// TIA Portal V20 export
// export: Created 2025-12-01T14:56:22.6904925Z, ExportSetting None, DisplayName Totally Integrated Automation Portal, DisplayVersion V20 Update 3, DisplayName TIA Portal Openness, DisplayVersion V20 Update 3, DisplayName TIA Portal Version Control Interface, DisplayVersion V20 Update 3, DisplayName STEP 7 Professional, DisplayVersion V20 Update 3, DisplayName STEP 7 Safety, DisplayVersion V20 Update 2, DisplayName WinCC Basic/Comfort/Advanced, DisplayVersion V20 Update 3, DisplayName WinCC Professional, DisplayVersion V20 Update 3, DisplayName WinCC Unified, DisplayVersion V20 Update 3
TYPE "MoviManualMesa_Eraman"
   STRUCT
      Avance_Rod : Bool;
      Retroceso_Rod : Bool;
      Avance_Cad_TR1 : Bool;
      Retroceso_Cad_TR1 : Bool;
      Subir_TR1 : Bool;
      Bajar_TR1 : Bool;
      Subir_TP1 : Bool;
      Bajar_TP1 : Bool;
      Avance_Cad_TR2 : Bool;
      Retroceso_Cad_TR2 : Bool;   // ...
      Subir_TR2 : Bool;   // ...
      Bajar_TR2 : Bool;   // ...
      Subir_TP2 : Bool;   // ...
      Bajar_TP2 : Bool;   // ...
      Subir_TPS3 : Bool;   // ...
      Bajar_TPS3 : Bool;   // ...
      Subir_TPE1 : Bool;   // ...
      Bajar_TPE1 : Bool;   // ...
      Byte2_bit2 : Bool;   // ...
      Byte2_bit3 : Bool;   // ...
      Byte2_bit4 : Bool;   // ...
      Byte2_bit5 : Bool;   // ...
      Byte2_bit6 : Bool;   // ...
      Byte2_bit7 : Bool;   // ...
      Avance_Cad_Ambos_Transfers : Bool;   // ...
      Retroceso_Cad_Ambos_Transfers : Bool;   // ...
      "Avance+Siguiente_Cad_TR1" : Bool;   // ...
      "Retroceso+Siguiente_Cad_TR1" : Bool;   // ...
      "Avance+Anterior_Cad_TR1" : Bool;   // ...
      "Retroceso+Anterior_Cad_TR1" : Bool;   // ...
      "Avance+Siguiente_Cad_TR2" : Bool;   // ...
      "Retroceso+Siguiente_Cad_TR2" : Bool;   // ...
      "Avance+Anterior_Cad_TR2" : Bool;   // ...
      "Retroceso+Anterior_Cad_TR2" : Bool;   // ...
      "Avance+Siguiente_Cad_Ambos_TR" : Bool;   // ...
      "Retroceso+Siguiente_Cad_Ambos_TR" : Bool;   // ...
      "Avance+Anterior_Cad_Ambos_TR" : Bool;   // ...
      "Retroceso+Anterior_Cad_Ambos_TR" : Bool;   // ...
      Byte4_bit6 : Bool;   // ...
      Byte4_bit7 : Bool;   // ...
      Byte5_bit0 : Bool;   // ...
      Byte5_bit1 : Bool;   // ...
      Reset_Mesa : Bool;   // ...
      Rearme : Bool;   // ...
      Byte5_bit4 : Bool;   // ...
      Byte5_bit5 : Bool;   // ...
      Byte5_bit6 : Bool;   // ...
      Byte5_bit7 : Bool;   // ...
      Byte6_bit0 : Bool;   // ...
      Byte6_bit1 : Bool;   // ...
      Byte6_bit2 : Bool;   // ...
      Byte6_bit3 : Bool;   // ...
      Byte6_bit4 : Bool;   // ...
      Byte6_bit5 : Bool;   // ...
      Byte6_bit6 : Bool;   // ...
      Byte6_bit7 : Bool;   // ...
      Byte7_bit0 : Bool;   // ...
      Byte7_bit1 : Bool;   // ...
      Byte7_bit2 : Bool;   // ...
      Byte7_bit3 : Bool;   // ...
      Byte7_bit4 : Bool;   // ...
      Byte7_bit5 : Bool;   // ...
      Byte7_bit6 : Bool;   // ...
      Byte7_bit7 : Bool;   // ...
   END_STRUCT;
END_TYPE
